# EPICS substitutions: odmApp/Db/bkh_odm_li00.substitutions
file bkhAi_simple.db {
pattern
    {ADDR,     ATTR,      DESC,         PORT, EGU, EOFF,        ESLO, PREC,  LOLO,   LOW,  HIGH,  HIHI,     LLSV,      LSV,      HSV,     HHSV}
    {   0, :1:Spare, "Spare 1", $(M)_3012_01,  mA,  0.0, 0.000610370,    3,   0.0,    "",  19.5,  20.0,    MINOR, NO_ALARM,    MINOR,    MAJOR}
    {   1, :2:Spare, "Spare 2", $(M)_3012_01,  mA,  0.0, 0.000610370,    3,   0.0,    "",  19.5,  20.0,    MINOR, NO_ALARM,    MINOR,    MAJOR}
}

file bkh_odm_common.db {
{None}
}
